{attribute 'enable_dynamic_creation'}
TYPE ST_HASHMAP_BUCKET_NODE EXTENDS ST_MAP_ENTRY :
STRUCT
	pNext : POINTER TO ST_HASHMAP_BUCKET_NODE;
END_STRUCT
END_TYPE

(* stored: Version 1.1.0.1
   DUT ST_HASHMAP_BUCKET_NODE: Id {e422d76a-b67e-0637-30b9-212329333d39} *)
